// TIA Portal V18 export
FUNCTION_BLOCK "KeyenceSR1000Ctrl"   // FB1800, SCL
{ S7_Optimized_Access := 'FALSE' }
VERSION : 0.1
// stored: AutoNumber false, IsIECCheckEnabled false, SetENOAutomatically false, UDAEnableTagReadback false
   VAR_INPUT
      iI_Address { ExternalAccessible := 'False'; ExternalVisible := 'False'; ExternalWritable := 'False'} : Int;   // hardware first input address
      iO_Address : Int;   // hardware first Output address
      iSysRun : Bool;
      iReset : Bool;
      iAuto : Bool;
      iManual : Bool;
      iReTriggerLimitTimes : USInt := 3;
   END_VAR
   VAR_OUTPUT
      oReady : Bool;
      oComplete : Bool;
      oError : Bool;
      oErrorCode : UInt;
   END_VAR
   VAR_IN_OUT
      ioAutoTrigger : Bool;
   END_VAR
   VAR DB_SPECIFIC
      sHMI { S7_SetPoint := 'True'} : "RCS_KeyenceSR1000_HMI1";
      sCtrl : Struct
         Sequence : Int;
      END_STRUCT;
      sCurrentCode : String[128];
   END_VAR
   VAR
      sAtCurrentCode AT sCurrentCode : Array[-1..128] of Byte;
   END_VAR
   VAR DB_SPECIFIC
      sInData { S7_SetPoint := 'True'} : "RCS_KeyenceSR1000_Input1";
      sOutData { S7_SetPoint := 'True'} : "RCS_KeyenceSR1000_Output1";
      sAutoOld : Bool;
      sManualOld : Bool;
      sBusyTimeOut : Bool;
      sRunTimer { S7_SetPoint := 'True'} : TON_TIME;
      sBusyTimer { S7_SetPoint := 'True'} : TON_TIME;
      sFindCurrentPos { S7_SetPoint := 'True'} : Int;
   END_VAR
   VAR_TEMP
      tAny : Any;
      tAnyParameters AT tAny : Struct
         SyntaxID : Byte;
         DataType : Byte;
         RepetitionFactor : Int;
         DB_Number : Word;
         MemoryAreaAddress : DWord;
      END_STRUCT;
      tOffset : Int;
      tEmpty : DWord;
      tIndex : Int;
      tRetVal : Int;
   END_VAR
BEGIN
   REGION Description
   (*
   KEYENCE SR-1000 Reader Function Block
   ruhlamat Automation Technologies(Suzhou) Co.,Ltd
   Copyright(c) 2020.All rights reserved.
   -------------------------------------------------------------------------------------------
   NAME OF FUNCTION BLOCK:"SR-1000Ctrl"
   NUMBER OF FUNCTION BLOCK: FB4021
   FAMILY:ruhlamat PSL
   VERSION:V1.0
   AUTHOR:Qianfeng.Yang
   LAST CHANGE:06.05.2021 (DB)
   -------------------------------------------------------------------------------------------
   Date Name Activity
   06.29.2020 Created by Qianfeng.Yang(V1.0)
   -------------------------------------------------------------------------------------------
   *)
   (*
   Trigger method: Level trigger. Handshaking: Disabled

   When reading is successful#################################################
   1 "Read request" is set to ON (1).
   2 When "Read request" is set to ON (1), the SR-1000 Series starts reading,and then "TRG BUSY" is set to ON (1).
   3 When the code is read, its data is written into "Read Data." "TRG BUSY" is set to OFF (0), and "Read Complete" is set to ON (1).
   4 "Read request" is set to OFF (0).
   5 It is confirmed that "Read Complete" is ON (1), and then "Read Complete Clear" is set to ON (1).
   6 When "Read Complete Clear" is set to ON (1), "Read Complete" is set to OFF (0).
   7 It is confirmed that "Read Complete" is OFF (0), and then "Read Complete Clear" is set to OFF (0).

   When reading fails##########################################################
   1 "Read request" is set to ON (1).
   2 When "Read request" is set to ON (1), the SR-1000 Series starts reading,and then "TRG BUSY" is set to ON (1).
   3 "Read request" is set to OFF (0).
   4 The code could not be read, so "ERROR" is written to "Result Data." "201" is written to "Read Result Code." "TRG BUSY" is set to OFF (0), and "Read Complete" is set to ON (1).
   5 It is confirmed that "Read Complete" is ON (1), and then "Read Complete Clear" is set to ON (1).
   6 When "Read Complete Clear" is set to ON (1), "Read Complete" and "Read Failure" are set to OFF (0).
   7 It is confirmed that "Read Complete" is OFF (0), and then "Read Complete Clear" is set to OFF (0).
   *)
   (*
   Error code List
     0=No error / (Reading success/operation succes)
   201=Reading error
   202=Comparison error / (The read code does not match the preset data)
   210=Tuning failure(Symbol unclear) / (The code could not be found within the field of)
   213=Tuning failure(Aborted) / (Tuning was aborted midwayview while tuning.)
   120=Control instruction receptionerror / (Another operation instruction was received during operation. (Operation instruction is notcompleted.)
   102=Bank No. error / (The bank number specification is invalid(other than 1 to 16))
   220=Preset data error / (Preset data specification is invalid.(Specified size is outside the range.))
   230=PROFINET data update error / (Shortage of specified size (Result data and present data size is beyond the limit.))

   FB ERROR
   1205=Failed to read HW Input data
   1206=Failed to write HW Output data
   1303=PG Running Timeout
   *)
   END_REGION

   (*Begin*)
   (*Read Data from KEYENCE SR-1000 TO PLC memory*)
   REGION Read inputs    
       #tAnyParameters.SyntaxID := 16#10;
       #tAnyParameters.DataType := 16#02;//Data type:Byte
       #tOffset := #iI_Address;
       #tAnyParameters.RepetitionFactor := 1;
       #tAnyParameters.DB_Number := 16#0;
       #tAnyParameters.MemoryAreaAddress := 16#8100_0000 OR (SHL(IN := INT_TO_DWORD(#tOffset), N := 3)); //B#16#81 Input Area
       IF BLKMOV(SRCBLK := #tAny, DSTBLK => #sInData.HandshakeAndGeneralErrorStatus) <> 0 THEN
           #sHMI.Status.Error := 1;
           #sHMI.Status.ErrorCode := 1205;
           GOTO Error;
       END_IF;
       #tOffset += #tAnyParameters.RepetitionFactor;
       #tAnyParameters.RepetitionFactor := 1;
       #tAnyParameters.MemoryAreaAddress := 16#8100_0000 OR (SHL(IN := INT_TO_DWORD(#tOffset), N := 3));
       IF BLKMOV(SRCBLK := #tAny, DSTBLK => #sInData.BusyStatus) <> 0 THEN
           #sHMI.Status.Error := 1;
           #sHMI.Status.ErrorCode := 1205;
           GOTO Error;
       END_IF;
       #tOffset += #tAnyParameters.RepetitionFactor;
       #tAnyParameters.RepetitionFactor := 1;
       #tAnyParameters.MemoryAreaAddress := 16#8100_0000 OR (SHL(IN := INT_TO_DWORD(#tOffset), N := 3));
       IF BLKMOV(SRCBLK := #tAny, DSTBLK => #sInData.CompletionStatus) <> 0 THEN
           #sHMI.Status.Error := 1;
           #sHMI.Status.ErrorCode := 1205;
           GOTO Error;
       END_IF;
       #tOffset += #tAnyParameters.RepetitionFactor;
       #tAnyParameters.RepetitionFactor := 1;
       #tAnyParameters.MemoryAreaAddress := 16#8100_0000 OR (SHL(IN := INT_TO_DWORD(#tOffset), N := 3));
       IF BLKMOV(SRCBLK := #tAny, DSTBLK => #sInData.ErrorStatus) <> 0 THEN
           #sHMI.Status.Error := 1;
           #sHMI.Status.ErrorCode := 1205;
           GOTO Error;
       END_IF;
       #tOffset += #tAnyParameters.RepetitionFactor;
       #tAnyParameters.RepetitionFactor := 1;
       #tAnyParameters.MemoryAreaAddress := 16#8100_0000 OR (SHL(IN := INT_TO_DWORD(#tOffset), N := 3));
       IF BLKMOV(SRCBLK := #tAny, DSTBLK => #sInData.TerminalStatus) <> 0 THEN
           #sHMI.Status.Error := 1;
           #sHMI.Status.ErrorCode := 1205;
           GOTO Error;
       END_IF;
       #tOffset += #tAnyParameters.RepetitionFactor;
       #tAnyParameters.RepetitionFactor := 1;
       #tAnyParameters.MemoryAreaAddress := 16#8100_0000 OR (SHL(IN := INT_TO_DWORD(#tOffset), N := 3));
       IF BLKMOV(SRCBLK := #tAny, DSTBLK => #sInData.UnstableReadStatus) <> 0 THEN
           #sHMI.Status.Error := 1;
           #sHMI.Status.ErrorCode := 1205;
           GOTO Error;
       END_IF;
       #tOffset += #tAnyParameters.RepetitionFactor;
       #tAnyParameters.RepetitionFactor := 8;
       #tAnyParameters.MemoryAreaAddress := 16#8100_0000 OR (SHL(IN := INT_TO_DWORD(#tOffset), N := 3));
       IF BLKMOV(SRCBLK := #tAny, DSTBLK => #sInData.MatchingLevelAndTotalEvaluationGradeStatus) <> 0 THEN
           #sHMI.Status.Error := 1;
           #sHMI.Status.ErrorCode := 1205;
           GOTO Error;
       END_IF;
       #tOffset += #tAnyParameters.RepetitionFactor;
       #tAnyParameters.RepetitionFactor := 20;
       #tAnyParameters.MemoryAreaAddress := 16#8100_0000 OR (SHL(IN := INT_TO_DWORD(#tOffset), N := 3));
       IF BLKMOV(SRCBLK := #tAny, DSTBLK => #sInData.OperationResultStatus) <> 0 THEN
           #sHMI.Status.Error := 1;
           #sHMI.Status.ErrorCode := 1205;
           GOTO Error;
       END_IF;
       #tOffset += #tAnyParameters.RepetitionFactor;
       #tAnyParameters.RepetitionFactor := 136;
       #tAnyParameters.MemoryAreaAddress := 16#8100_0000 OR (SHL(IN := INT_TO_DWORD(#tOffset), N := 3));
       IF BLKMOV(SRCBLK := #tAny, DSTBLK => #sInData.ReadData) <> 0 THEN
           #sHMI.Status.Error := 1;
           #sHMI.Status.ErrorCode := 1205;
           GOTO Error;
       END_IF;
   END_REGION ;

   (*Status*)
   REGION Status
       (*Set String length*)
       #sAtCurrentCode[-1] := 128;

       (*Ready*)
       #sHMI.Status.Ready := #iSysRun AND #sCtrl.Sequence = 0
       AND NOT #sInData.BusyStatus.TrggerBusy
       AND NOT #sInData.HandshakeAndGeneralErrorStatus.Error
       AND NOT #sInData.CompletionStatus.ReadComplete
       AND NOT #sInData.ErrorStatus.ReadFailure
       AND NOT #sHMI.Status.Error;//20210605

       (*Busy*)
       #sHMI.Status.Busy := #sInData.BusyStatus.TrggerBusy;

       (*Failure*)
       #sHMI.Status.Failure := #sInData.ErrorStatus.ReadFailure;

       (*Timeout*)
       #sRunTimer(IN := #sCtrl.Sequence <> 0 OR NOT #sHMI.Status.Ready,
                  PT := T#3000MS,
                  Q => #sHMI.Status.TimeOut);
       #sBusyTimer(IN := #sInData.BusyStatus.TrggerBusy,
               PT := T#1000MS,
               Q => #sBusyTimeOut); //20210605

       (*SR1000 Error and Error Code*)    
       IF #sInData.HandshakeAndGeneralErrorStatus.Error THEN
           #sHMI.Status.Error := 1;
           #sHMI.Status.ErrorCode := #sInData.OperationResultStatus.ReadResultCode;
       ELSIF #sHMI.Status.TimeOut THEN
           #sHMI.Status.Error := 1;
           #sHMI.Status.ErrorCode := 1303;
           #sOutData.OperationInstructionControl.ReadRequest := 0; //20210605
       END_IF;



       (*HMI Display*)
       #sHMI.Status.Sequence := #sCtrl.Sequence;

       #sHMI.Indata.ReadComplete := #sInData.CompletionStatus.ReadComplete;
       #sHMI.Indata.ReadFailure := #sInData.ErrorStatus.ReadFailure;
       #sHMI.Indata.GeneralErrorCode := #sInData.OperationResultStatus.GeneralErrorCode;
       #sHMI.Indata.ReadResultCode := #sInData.OperationResultStatus.ReadResultCode;
       #sHMI.Indata.ResultDataSize := #sInData.ReadData.ResultDataSize;

       #sHMI.Outdata.ReadCompleteClear := #sOutData.CompletionClearControl.ReadCompleteClear;
       #sHMI.Outdata.ErrorClear := #sOutData.LatchAndErrorClearControl.ErrorClear;
       #sHMI.Outdata.ReadRequest := #sOutData.OperationInstructionControl.ReadRequest;

   END_REGION ;
   (*Control*)
   REGION Control
       (*Reset command*)
       IF NOT #iSysRun OR (#iManual XOR #sManualOld) OR (#iAuto XOR #sAutoOld) THEN
           #sHMI.Manual.Trigger := 0;
           #ioAutoTrigger := 0;
           #sHMI.Status.iReTriggerTimes := 0;
           #sOutData.OperationInstructionControl.ReadRequest := 0; //20210605
       END_IF;
       #sManualOld := #iManual;
       #sAutoOld := #iAuto;


       //Control Sequece************************************************************************)
       CASE #sCtrl.Sequence OF
           0:(*Trigger*)
               #sOutData.CompletionClearControl.ReadCompleteClear := #sInData.CompletionStatus.ReadComplete;
               IF #sHMI.Status.Ready AND ((#iAuto AND #ioAutoTrigger) XOR (#iManual AND #sHMI.Manual.Trigger)) THEN
                   #sHMI.Status.LastCode := #sHMI.Status.CurrentCode;
                   #sHMI.Status.CurrentCode := '';
                   #sHMI.Status.CurrentLength := 0;
                   #sHMI.Status.ReadOk := 0;
                   #sHMI.Status.ReadNok := 0;
                   #sHMI.Status.Complete := 0;
                   #sOutData.OperationInstructionControl.ReadRequest := 1; //Trigger
                   #sOutData.CompletionClearControl.ReadCompleteClear := 0;
                   #sCtrl.Sequence := 1;
               ELSE
                   #sOutData.OperationInstructionControl.ReadRequest := 0;
               END_IF;
           1:(*Reading*)
               IF NOT #sInData.HandshakeAndGeneralErrorStatus.Error
                   AND #sOutData.OperationInstructionControl.ReadRequest
                   AND #sInData.BusyStatus.TrggerBusy THEN
                   #sHMI.Status.iReTriggerTimes := #sHMI.Status.iReTriggerTimes + 1;
                   //#sHMI.Manual.Trigger := 0;
                   #sCtrl.Sequence := 2;
               END_IF;
           2:(*Complete*)
               IF (NOT #sInData.HandshakeAndGeneralErrorStatus.Error AND NOT #sInData.BusyStatus.TrggerBusy AND #sInData.CompletionStatus.ReadComplete)
                   OR #sBusyTimeOut THEN
                   #sOutData.OperationInstructionControl.ReadRequest := 0;
                   #sCtrl.Sequence := 3;
               END_IF;
           3:(*Result*)
               IF NOT #sInData.HandshakeAndGeneralErrorStatus.Error
                   AND NOT #sOutData.OperationInstructionControl.ReadRequest
                   AND #sInData.CompletionStatus.ReadComplete
                   AND #sInData.ReadData.ResultDataSize <= 128
                   AND #sInData.ReadData.ResultDataSize > 0 THEN
                   Chars_TO_Strg(Chars := #sInData.ReadData.ResultData,
                                 pChars := 0, //20210605
                                 Cnt := #sInData.ReadData.ResultDataSize,
                                 Strg => #sCurrentCode);

                   #sFindCurrentPos  :=  FIND(IN1 := #sCurrentCode, IN2 := '$R');

                   #sCurrentCode := DELETE(IN := #sCurrentCode, L := 2, P := #sFindCurrentPos);

                   #sHMI.Status.CurrentCode := #sCurrentCode;
                   IF #sHMI.Status.CurrentCode = 'ERROR' OR #sInData.ErrorStatus.ReadFailure THEN
                       #sCtrl.Sequence := 4;
                   ELSE
                       #sHMI.Status.ReadOk := 1;
                       #sHMI.Status.ReadNok := 0;
                       #sCtrl.Sequence := 5;
                   END_IF;
               END_IF;

           4: (*ReTrigger*)
               IF #sHMI.Status.iReTriggerTimes < #iReTriggerLimitTimes THEN
                   #sOutData.CompletionClearControl.ReadCompleteClear := 1;
                   IF NOT #sInData.CompletionStatus.ReadComplete AND NOT #sInData.ErrorStatus.ReadFailure THEN
                       #sCtrl.Sequence := 0;
                   END_IF;
               ELSE
                   #sHMI.Status.ReadOk := 0;
                   #sHMI.Status.ReadNok := 1;
                   #sCtrl.Sequence := 5;
               END_IF;

           5:(*Clear*)
               IF NOT #sOutData.OperationInstructionControl.ReadRequest
                   AND #sInData.CompletionStatus.ReadComplete THEN
                   #sOutData.CompletionClearControl.ReadCompleteClear := 1;
               ELSE
                   #sOutData.CompletionClearControl.ReadCompleteClear := 0;
                   #ioAutoTrigger := 0;
                   #sHMI.Manual.Trigger := 0;
                   #sHMI.Status.iReTriggerTimes := 0;
                   #sHMI.Status.Complete := 1;
                   #sCtrl.Sequence := 0;
               END_IF;
           ELSE(*Limit*)
               #sCtrl.Sequence := 0;
       END_CASE;
   END_REGION ;

   REGION Reset
   IF (#sHMI.Status.Error OR #sHMI.Status.Failure OR #sHMI.Status.TimeOut) THEN
       IF #iReset THEN
           #sOutData.LatchAndErrorClearControl.ErrorClear := 1;
           #sOutData.OperationInstructionControl.ReadRequest := 0;
           #ioAutoTrigger := 0;
           #sHMI.Manual.Trigger := 0;
           #sCtrl.Sequence := 0;
           #sHMI.Status.Error := 0;
           #sHMI.Status.ErrorCode := 0;
       END_IF;
   ELSE
       #sOutData.LatchAndErrorClearControl.ErrorClear := 0;
   END_IF;
   END_REGION ;


   (*Write Data from PLC memory to KEYENCE SR-1000*)
   REGION Write outputs
       #tAnyParameters.SyntaxID := 16#10;
       #tAnyParameters.DataType := 16#02;
       #tOffset := #iO_Address;
       #tAnyParameters.RepetitionFactor := 1;
       #tAnyParameters.DB_Number := 16#0;
       #tAnyParameters.MemoryAreaAddress := 16#8200_0000 OR (SHL(IN := INT_TO_DWORD(#tOffset), N := 3)); //B#16#82 Output Area
       IF BLKMOV(SRCBLK := #sOutData.LatchAndErrorClearControl, DSTBLK => #tAny) <> 0 THEN
           #sHMI.Status.Error := 1;
           #sHMI.Status.ErrorCode := 1206;
           GOTO Error;
       END_IF;
       #tOffset += #tAnyParameters.RepetitionFactor;
       #tAnyParameters.RepetitionFactor := 1;
       #tAnyParameters.MemoryAreaAddress := 16#8200_0000 OR (SHL(IN := INT_TO_DWORD(#tOffset), N := 3));
       IF BLKMOV(SRCBLK := #sOutData.OperationInstructionControl, DSTBLK => #tAny) <> 0 THEN
           #sHMI.Status.Error := 1;
           #sHMI.Status.ErrorCode := 1206;
           GOTO Error;
       END_IF;
       #tOffset += #tAnyParameters.RepetitionFactor;
       #tAnyParameters.RepetitionFactor := 1;
       #tAnyParameters.MemoryAreaAddress := 16#8200_0000 OR (SHL(IN := INT_TO_DWORD(#tOffset), N := 3));
       IF BLKMOV(SRCBLK := #sOutData.CompletionClearControl, DSTBLK => #tAny) <> 0 THEN
           #sHMI.Status.Error := 1;
           #sHMI.Status.ErrorCode := 1206;
           GOTO Error;
       END_IF;
       #tOffset += #tAnyParameters.RepetitionFactor;
       #tAnyParameters.RepetitionFactor := 2;
       #tAnyParameters.MemoryAreaAddress := 16#8200_0000 OR (SHL(IN := INT_TO_DWORD(#tOffset), N := 3));
       IF BLKMOV(SRCBLK := #sOutData.ParameterBankNumber, DSTBLK => #tAny) <> 0 THEN
           #sHMI.Status.Error := 1;
           #sHMI.Status.ErrorCode := 1206;
           GOTO Error;
       END_IF;
       #tOffset += #tAnyParameters.RepetitionFactor;
       #tAnyParameters.RepetitionFactor := 130;
       #tAnyParameters.MemoryAreaAddress := 16#8200_0000 OR (SHL(IN := INT_TO_DWORD(#tOffset), N := 3));
       IF BLKMOV(SRCBLK := #sOutData.UserData, DSTBLK => #tAny) <> 0 THEN
           #sHMI.Status.Error := 1;
           #sHMI.Status.ErrorCode := 1206;
           GOTO Error;
       END_IF;

   //FB OUTPUT    
       #oReady := #sHMI.Status.Ready;
       #oComplete := #sHMI.Status.Complete;
       #oError := #sHMI.Status.Error;
       #oErrorCode := #sHMI.Status.ErrorCode;

   END_REGION ;
   (*The end of the function block*)
   REGION End function
       ENO := 1;
       RETURN;
   Error:
       #sHMI.Status.Ready := 0;
       #tEmpty := 16#0000_0000;
       #tRetVal := FILL(BVAL := #tEmpty, BLK => #sOutData.LatchAndErrorClearControl);
       #tRetVal := FILL(BVAL := #tEmpty, BLK => #sOutData.OperationInstructionControl);
       #tRetVal := FILL(BVAL := #tEmpty, BLK => #sOutData.CompletionClearControl);
       #tRetVal := FILL(BVAL := #tEmpty, BLK => #sOutData.ParameterBankNumber);
       #tRetVal := FILL(BVAL := #tEmpty, BLK => #sOutData.UserData);
       ENO := 0;
       RETURN;
   END_REGION ;
END_FUNCTION_BLOCK
